TYPE
    ST_Manual_Allocated :
    STRUCT
        OutRobot       : ST_Manual_OutRobot;       // Allocated out robot manual control
        NeedleRobot    : ST_Manual_NeedleRobot; // Allocated allocated robot manual control
        Allocate       : ST_Manual_Allocate;      // Allocated round belt manual control
        TurnTable      : ST_Manual_TurnTable;      // Allocated turn table manual control
        PullOutCV      : ST_Manual_PullOutCV;        // Allocated pullout conveyor manual control
        TransCV        : ST_Manual_TransCV;        // Allocated transmit conveyor manual control
    END_STRUCT
END_TYPE

(* stored: Version 1.1.0.1, ProductVersion 3.1.4024.13
   DUT ST_Manual_Allocated: Id {1d8017de-800a-4470-8d32-c95047e9e9a7} *)
